INTERFACE I_Value

END_INTERFACE

(* stored: Version 1.1.0.1
   Itf I_Value: Id {11eb2c2c-756a-4a5b-9fbd-9cf867ad8056} *)
